{attribute 'linkalways'} 
{attribute 'no_explicit_call' := 'This FB is a CLASS and must be accessed using methods or properties'}
{attribute 'enable_dynamic_creation'}
FUNCTION_BLOCK ChunkableServerResponse IMPLEMENTS I_ServerResponse
VAR
	serverResponse : I_ServerResponse;
	chunkedResponseManager : I_ChunkedResponseManager;
END_VAR

METHOD PUBLIC Accepted
VAR_INPUT
END_VAR
serverResponse.Accepted();
END_METHOD

METHOD PUBLIC Busy
VAR_INPUT
END_VAR
serverResponse.Busy();
END_METHOD

METHOD PUBLIC Error
VAR_INPUT
	ErrorCode : T_MAXSTRING;
	Message : T_MAXSTRING;
END_VAR
serverResponse.Error(ErrorCode, Message);
END_METHOD

METHOD FB_init : BOOL
VAR_INPUT
	bInitRetains : BOOL; // if TRUE, the retain variables are initialized (warm start / cold start)
	bInCopyCode : BOOL;  // if TRUE, the instance afterwards gets moved into the copy code (online change)
	ServerResponse : I_ServerResponse;
	ChunkedResponseManager : I_ChunkedResponseManager;
END_VAR
THIS^.serverResponse := ServerResponse;
This^.chunkedResponseManager := ChunkedResponseManager;
END_METHOD

PROPERTY PUBLIC Header : I_Header
GET
Header := serverResponse.Header;
END_GET
END_PROPERTY

PROPERTY PUBLIC HeadersSent : BOOL
GET
HeadersSent := serverResponse.HeadersSent;
END_GET
END_PROPERTY

METHOD PUBLIC Pending
VAR_INPUT
	ResponseId : REFERENCE TO T_MAXSTRING;
	RetryDelayInMs : UDINT;
END_VAR
serverResponse.Pending(ResponseId, RetryDelayInMs);
END_METHOD

METHOD PUBLIC Success
VAR_INPUT
END_VAR
serverResponse.Success();
END_METHOD

METHOD PUBLIC SuccessWithPayload
VAR_INPUT
	PayloadDataAddress : PVOID;
	PayloadDataSize : UDINT;
END_VAR
chunkedResponseManager.HandleSuccessWithPayload(serverResponse, PayloadDataAddress, PayloadDataSize);
END_METHOD

END_FUNCTION_BLOCK

(* stored: Version 1.1.0.1, ProductVersion 3.1.4024.15
   POU ChunkableServerResponse: Id {2fe2454c-a3f1-0dae-05f0-d9a275bb7efe}, SpecialFunc None
   Folder Constructor: Id {97f632d6-5e51-040c-3eb1-fe42fade6fe1}
   Method Accepted: Id {a7354322-c96d-0504-03f0-8a61280228f7}
   Method Busy: Id {dc194327-1054-09c4-1d3c-a5bd62a06f5f}
   Method Error: Id {cdb1f046-0dbf-0f4a-1a04-825152a18feb}
   Method FB_init: Id {f147299a-b64c-085b-1319-2bb7394bb5ef}
   Property Header: Id {b4164af5-e8d3-04a2-0204-ce4113b939bb}
   Get Get: Id {ddcd17fb-7a3a-040d-3c52-6398234501c9}
   Property HeadersSent: Id {f3778ec9-42cd-0ec9-0dac-4d3a79b8686f}
   Get Get: Id {476cd823-6b65-0c7f-23d4-14c7c4e5db37}
   Method Pending: Id {aedde6f8-2a14-001e-1c13-aa18243a34cb}
   Method Success: Id {ffdac1be-9606-0956-036c-ef54603ebe09}
   Method SuccessWithPayload: Id {27433e92-5bf9-0fd0-048b-a68ac0f6f956} *)
